FUNCTION_BLOCK STRIP4 (* 4-Pen Strip Chart Recorder *)
  (* Standard: 61499-1; Classification: Service Interface; ApplicationDomain: Human Interface; Function: Recorder; Type: Strip Chart *)
  (* Version 0.1, 2004-09-03, JHC, Rockwell Automation, Deleted QI, QO, MAX_SCALE, MIN_SCALE; made inputs UINT{0..100}. *)
  (* Compiler header: package fb.rt.swing; *)
  (* Compiler classdef: public class STRIP4 extends STRIP3 *)
  (* Compiler Java IBM VisualAge 3.0 *)
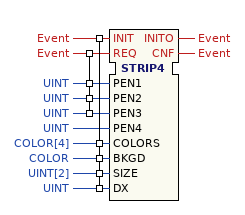
  EVENT_INPUT
    INIT WITH COLORS, BKGD, SIZE, DX;
    REQ WITH PEN1, PEN2, PEN3;
  END_EVENT
  EVENT_OUTPUT
    INITO;
    CNF;
  END_EVENT
  VAR_INPUT
    PEN1 : UINT; (* Pen 1 Position, 0-100% *)
    PEN2 : UINT; (* Pen 2 Position, 0-100% *)
    PEN3 : UINT; (* Pen 3 Position, 0-100% *)
    PEN4 : UINT; (* Pen 4 Position, 0-100% *)
    COLORS : ARRAY [0..3] OF COLOR := [red,blue,green,yellow]; (* PEN1,2,3,4 Colors *)
    BKGD : COLOR := lightGray; (* Background Color *)
    SIZE : ARRAY [0..1] OF UINT := [200,200]; (* Width,Height *)
    DX : UINT := 10; (* x-increment size *)
  END_VAR
END_FUNCTION_BLOCK
